Yaskawa INFORM job: MASTER_BATMAN_R2.JBI

/JOB
//NAME MASTER_BATMAN_R2
///FOLDERNAME MASTER-SCIANA-R2
//POS
///NPOS 7,7,7,0,0,0
///TOOL 0
///POSTYPE PULSE
///PULSE
C00000=-5026,39564,34271,3752,88090,-85590
C00001=-5026,38657,30797,3753,89758,-85540
C00002=-5026,38657,30797,3753,89758,-52778
C00003=-5643,130418,55957,-12263,93447,23906
C00004=-10129,1594,-22592,15665,55683,74718
C00005=-16138,-42092,-35388,10444,39088,-86293
C00006=-5026,39564,34271,3752,88090,-85590
BC00000=62200,677985,1036994
BC00001=62200,669168,820015
BC00002=62200,669168,1028696
BC00003=66423,1186109,1064960
BC00004=50954,978615,1075052
BC00005=126121,734025,1068204
BC00006=62200,677985,1036994
EC00000=0,556475
EC00001=798157,1112952
EC00002=798157,1112952
EC00003=363194,1107221
EC00004=798157,1112952
EC00005=798157,1112952
EC00006=0,556475
//INST
///DATE 2024/07/31 08:18
///ATTR SC,RW
///GROUP1 RB1,BS1
///GROUP2 ST1
NOP
MOVJ C00000 BC00000 VJ=100.00  +MOVJ EC00000 VJ=100.00
MOVJ C00001 BC00001 VJ=100.00  +MOVJ EC00001 VJ=100.00
PAUSE
PAUSE
'SCIAGNIJ USZY ZE SCIANY
MOVJ C00002 BC00002 VJ=100.00  +MOVJ EC00002 VJ=100.00
MOVJ C00003 BC00003 VJ=100.00  +MOVJ EC00003 VJ=100.00
CALL JOB:BATMAN_ALL2
MOVJ C00004 BC00004 VJ=50.00  +MOVJ EC00004 VJ=50.00
CALL JOB:BATMAN_2STR2
MOVJ C00005 BC00005 VJ=50.00  +MOVJ EC00005 VJ=50.00
CALL JOB:BATMAN_4SPOINY2
MOVJ C00006 BC00006 VJ=100.00  +MOVJ EC00006 VJ=100.00
PAUSE
END
